FUNCTION_BLOCK AIWS_PUBLISH_1 (* Publish a WSTRING from an AIWS adapter to one or many SUBSCRIBE_1 Blocks, buffered with a D_FF *)
  (* Standard: 61499-2; Description: Copyright (c) 2026 HR Agrartechnik GmbH This program and the accompanying materials are made available under the terms of the Eclipse Public License 2.0 which is available at https://www.eclipse.org/legal/epl-2.0/ SPDX-License-Identifier: EPL-2.0 *)
  (* Version 1.0, 2026-08-07, Franz Höpfinger, HR Agrartechnik GmbH, initial API and implementation and/or initial documentation *)
  PACKAGE adapter::net;
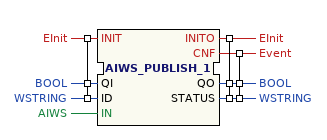
  EVENT_INPUT
    INIT : EInit WITH QI, ID; (* Initialization *)
  END_EVENT
  EVENT_OUTPUT
    INITO : EInit WITH QO, STATUS; (* Initialization Confirm *)
    CNF WITH QO, STATUS; (* Data was sent *)
  END_EVENT
  VAR_INPUT
    QI : BOOL;
    ID : WSTRING;
  END_VAR
  VAR_OUTPUT
    QO : BOOL;
    STATUS : WSTRING;
  END_VAR
  SOCKETS
    IN : adapter::types::unidirectional::AIWS; (* WSTRING to publish *)
  END_SOCKETS
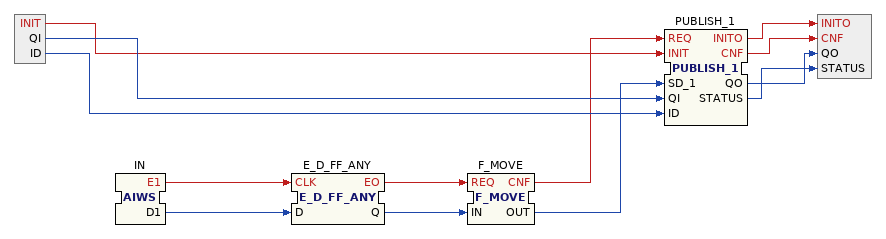
  FBS
    E_D_FF_ANY : iec61499::events::E_D_FF_ANY;
    F_MOVE : iec61131::selection::F_MOVE; {SET_ATTRIBUTE(DataType, WSTRING)}
    PUBLISH_1 : iec61499::net::PUBLISH_1;
  END_FBS
  EVENT_CONNECTIONS
    PUBLISH_1.INITO TO INITO;
    PUBLISH_1.CNF TO CNF;
    IN.E1 TO E_D_FF_ANY.CLK;
    E_D_FF_ANY.EO TO F_MOVE.REQ;
    F_MOVE.CNF TO PUBLISH_1.REQ;
    INIT TO PUBLISH_1.INIT;
  END_CONNECTIONS
  DATA_CONNECTIONS
    PUBLISH_1.QO TO QO;
    PUBLISH_1.STATUS TO STATUS;
    IN.D1 TO E_D_FF_ANY.D;
    E_D_FF_ANY.Q TO F_MOVE.IN;
    F_MOVE.OUT TO PUBLISH_1.SD_1;
    QI TO PUBLISH_1.QI;
    ID TO PUBLISH_1.ID;
  END_CONNECTIONS
END_FUNCTION_BLOCK
